PROGRAM P_Demo_FB_PN_IM3_WRITE
VAR
    fbIM3Write    : FB_PN_IM3_WRITE;
    bWriteDesc    : BOOL := FALSE;            // 在线上升沿触发写入
    sDescriptor   : STRING(54) := 'CfgRev=2.3 maint by EE-team';   // 待写描述
    bBusy         : BOOL;
    bErr          : BOOL;
    nErrId        : UDINT;
END_VAR

// ============================================================
// Tc2_ProfinetDiag.FB_PN_IM3_WRITE 演示程序
// ============================================================
// 场景：给设备写 I&M3 自定义描述。
// 价值：设备自带注释，免外部映射。
// 验证：登录后 bWriteDesc 上升沿写入 sDescriptor。
// 验证步骤：
//   1. 右键 PLC 项目下 POUs 文件夹 → Add → Existing Item → 选本 .TcPOU 文件
//   2. 引用 Tc2_ProfinetDiag（References → Add library）
//   3. 编译 → 登录 → 运行；按上方『验证』指引在线写值观察
// ============================================================

// 把自定义描述写入设备 I&M3
fbIM3Write(
    bStart := bWriteDesc,
    NETID  := '',
    PORT   := 16#1001,
    st_IM_Descriptor := sDescriptor,
    bBusy  => bBusy,
    bError => bErr,
    iErrorID => nErrId
);

END_PROGRAM

(* stored: Version 1.1.0.1, ProductVersion 3.1.4024.5
   POU P_Demo_FB_PN_IM3_WRITE: Id {8cde2c42-d1c8-57d1-bc7f-524dfdac37d2}, SpecialFunc None *)
